GLOBALCONSTANTS SubStrings (* Global constants *)
  (* Standard: 61499-1 *)
  (* Version 1.0, 2026-10-05, Franz Höpfinger, Meisterschulen am Ostbahnhof *)
  PACKAGE Meins::Servo_Slider_OPC;
  VAR_GLOBAL CONSTANT
    SERVO_Q2_ANGLE_SET : WSTRING := "opc_ua[READ;/Objects/Servo/Q02/ANGLE_SET,1:s=SERVO_Q2_ANGLE_SET]";
    SERVO_Q2_ANGLE : WSTRING := "opc_ua[WRITE;/Objects/Servo/Q02/ANGLE,1:s=SERVO_Q2_ANGLE]";
  END_VAR
END_GLOBALCONSTANTS
